Fanuc KAREL source: w_grp1.kl

PROGRAM w_grp1
%NOLOCKGROUP
VAR
  p : POSITION
  q : POSITION
  i : INTEGER
  r : REAL
BEGIN
  WITH $GROUP[1].$SPEED = 500, $GROUP[1].$MOTYPE = i MOVE TO p
END w_grp1
